// TIA Portal project "s14_code" (V21)

(* hardware
DEVICE "S7-1500/ET200MP station_1"  S7-1500 station
   slot 0: "Rail_0"  Rack  6ES7 590-1***0-0AA0
   slot 1: "ZZPLC"  CPU 1511-1 PN  6ES7 511-1AK00-0AB0  V1.8
      slot 3: "CPU display_1"  6ES7591-1AA00-0AA0
      slot 32768: "PROFINET interface_1"  X1
         slot 32769: "Port_1"  X1 P1
         slot 32770: "Port_2"  X1 P2
*)

// ===== PLC "ZZPLC"  CPU 1511-1 PN =====
// protected blocks, not shown: "ZZSCL"

VAR_GLOBAL   // PLC tag table "Default tag table"
   "ZZALPHA" AT %M10.0 : Bool;
   "ZZB" AT %M10.1 : Bool;
   "ZZC" AT %M10.2 : Bool;
   "ZZOUT" AT %M11.0 : Bool;
   "ZZN1" AT %MW20 : Int;
   "ZZN2" AT %MW22 : Int;
   "ZZN3" AT %MW24 : Int;
END_VAR

DATA_BLOCK "ZZDATA"   // DB1
{ S7_Optimized_Access := 'TRUE' }
VERSION : 0.1
   VAR
      run : Bool;
      speed : Int;
   END_VAR
BEGIN
END_DATA_BLOCK

DATA_BLOCK "ZZFB_DB"   // DB3
{ S7_Optimized_Access := 'TRUE' }
VERSION : 0.1
// stored: InstanceOfName ZZFB
"ZZFB"
BEGIN
END_DATA_BLOCK

// folder: System blocks/Program resources

DATA_BLOCK "IEC_Timer_0_DB"   // DB2
{ S7_Optimized_Access := 'TRUE' }
AUTHOR : Simatic
FAMILY : IEC
NAME : IEC_TMR
VERSION : 1.0
// stored: InstanceOfName IEC_TIMER
"IEC_TIMER"
BEGIN
END_DATA_BLOCK

// folder: (top level)

FUNCTION_BLOCK "ZZFB"   // FB1, LAD
{ S7_Optimized_Access := 'TRUE' }
VERSION : 0.1
   VAR_INPUT
      in1 : Bool;
   END_VAR
   VAR_OUTPUT
      out1 : Bool;
   END_VAR
BEGIN

REGION Network 1
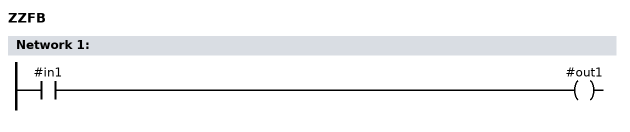
   RUNG wire#powerrail
      Contact( #in1 )
      Coil( #out1 )
   END_RUNG
   // the same network as SCL:
   #out1 := #in1;
END_REGION
END_FUNCTION_BLOCK

FUNCTION "ZZFBD" : Void   // FC1, FBD
{ S7_Optimized_Access := 'TRUE' }
VERSION : 0.1
BEGIN

REGION Network 1
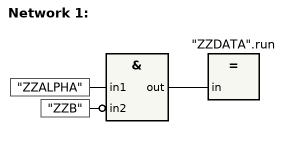
   "ZZDATA".run := "ZZALPHA" AND NOT "ZZB";
END_REGION
END_FUNCTION

FUNCTION "ZZSTL" : Void   // FC3, STL
{ S7_Optimized_Access := 'TRUE' }
VERSION : 0.1
BEGIN

REGION Network 1
         A     "ZZALPHA";
         AN    "ZZB";
         =     "ZZOUT";
END_REGION

REGION Network 2
         L     "ZZN1";
         L     5;
         +I;
         T     "ZZN3";
END_REGION
END_FUNCTION

ORGANIZATION_BLOCK "Main"   // OB1, LAD, ProgramCycle
TITLE = "Main Program Sweep (Cycle)"
{ S7_Optimized_Access := 'TRUE' }
VERSION : 0.1
   VAR_INPUT
      Initial_Call : Bool;   // Initial call of this OB
      Remanence : Bool;   // =True, if remanent data are available
   END_VAR
   VAR_TEMP   // added for the SCL form of the ladder/FBD networks
      _w1 : Bool;
      _w2 : Bool;
   END_VAR
BEGIN

REGION Network 1: ZZ series
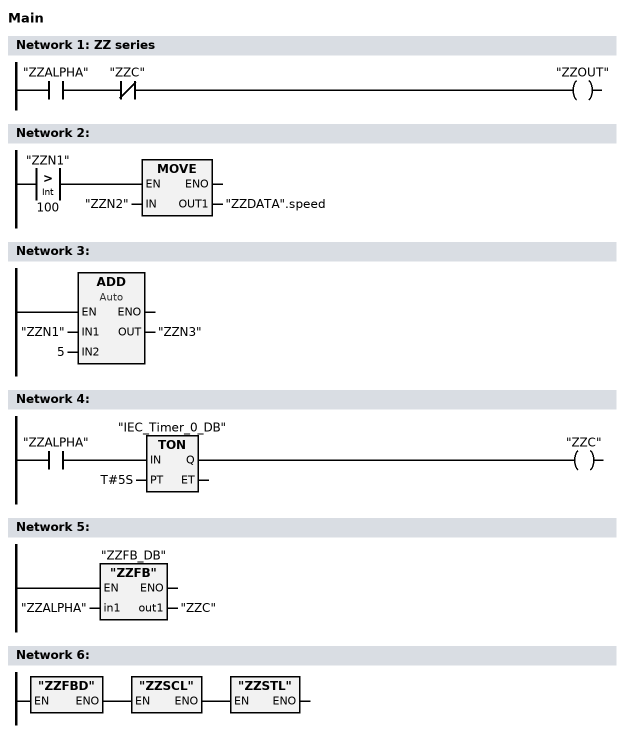
   RUNG wire#powerrail
      Contact( "ZZALPHA" )
      I_Contact( "ZZC" )
      Coil( "ZZOUT" )
   END_RUNG
   // the same network as SCL:
   "ZZOUT" := "ZZALPHA" AND NOT "ZZC";
END_REGION

REGION Network 2
   RUNG wire#powerrail
      { S7_Templates := "SrcType := Int" } GT_Contact(in1 := "ZZN1", in2 := 100)
      Move(in := "ZZN2", out1 => "ZZDATA".speed)
   END_RUNG
   // the same network as SCL:
   IF "ZZN1" > 100 THEN "ZZDATA".speed := "ZZN2"; END_IF;
END_REGION

REGION Network 3
   RUNG wire#powerrail
      Add(in1 := "ZZN1", in2 := 5, out => "ZZN3")
   END_RUNG
   // the same network as SCL:
   "ZZN3" := "ZZN1" + 5;
END_REGION

REGION Network 4
   "IEC_Timer_0_DB".TON(IN := "ZZALPHA", PT := T#5S);
   "ZZC" := "IEC_Timer_0_DB".Q;
END_REGION

REGION Network 5
   RUNG wire#powerrail
      "ZZFB_DB"(in1 := "ZZALPHA", out1 => "ZZC")
   END_RUNG
   // the same network as SCL:
   "ZZFB_DB"(in1 := "ZZALPHA", out1 => "ZZC");   // "ZZFB"
END_REGION

REGION Network 6
   RUNG wire#powerrail
      "ZZFBD"()
      "ZZSCL"()
      "ZZSTL"()
   END_RUNG
   // the same network as SCL:
   "ZZFBD"(ENO => #_w1);
   "ZZSCL"(EN := #_w1, ENO => #_w2);
   IF #_w2 THEN "ZZSTL"(); END_IF;
END_REGION
END_ORGANIZATION_BLOCK